// Mitsubishi GX Works2 project: SAPIR_SHELLY_FINAL   PLC: FX3G

// global labels: Global1
VAR_GLOBAL
  Start_Day_Light AT Y007 : BOOL;
  Input1 AT D1110 : REAL;
  Input2 AT D1120 : REAL;
  Input3 AT D1130 : REAL;
  Input4 AT D1140 : REAL;
  Raspberry AT D1115 : REAL;
  Lemon AT D1125 : REAL;
  Stability AT D1135 : REAL;
  Bears AT D1145 : REAL;
  Fin_inp AT M23 : BOOL;
  Startday AT X007 : BOOL;
  Stopday AT M27 : BOOL;
  AnalogOutput AT D8282 : INT;
  Package_Num AT D2000 : REAL;
  Emergency AT X005 : BOOL;
  Prepare_Flav AT X001 : BOOL;
  AnalogInput1 AT D8280 : INT;
END_VAR
VAR_GLOBAL CONSTANT
  Divide : REAL := 400.0;
END_VAR
VAR_GLOBAL
  DivOutput AT D1310 : REAL;
END_VAR
VAR_GLOBAL CONSTANT
  Regular_ice : REAL := 5.0;
END_VAR
VAR_GLOBAL
  Flav_Succeed AT M28 : BOOL;
  Regular_Chosen AT M30 : BOOL;
END_VAR
VAR_GLOBAL CONSTANT
  Needed1R : REAL := 280.0;
END_VAR
VAR_GLOBAL
  EnoughRas_R AT M29 : BOOL;
END_VAR
VAR_GLOBAL CONSTANT
  Needed2R : REAL := 455.0;
END_VAR
VAR_GLOBAL
  EnoughLem_R AT M40 : BOOL;
END_VAR
VAR_GLOBAL CONSTANT
  Needed3R : REAL := 105.0;
END_VAR
VAR_GLOBAL
  EnoughStab_R AT M41 : BOOL;
END_VAR
VAR_GLOBAL CONSTANT
  Needed4R : REAL := 28.0;
END_VAR
VAR_GLOBAL
  EnoughBear_R AT M42 : BOOL;
END_VAR
VAR_GLOBAL CONSTANT
  Needed1P : REAL := 385.0;
END_VAR
VAR_GLOBAL
  EnoughRas_P AT M45 : BOOL;
END_VAR
VAR_GLOBAL CONSTANT
  Needed2P : REAL := 665.0;
END_VAR
VAR_GLOBAL
  EnoughLem_P AT M48 : BOOL;
END_VAR
VAR_GLOBAL CONSTANT
  Needed3P : REAL := 210.0;
END_VAR
VAR_GLOBAL
  EnoughStab_P AT M50 : BOOL;
END_VAR
VAR_GLOBAL CONSTANT
  Needed4P : REAL := 70.0;
END_VAR
VAR_GLOBAL
  EnoughBear_P AT M52 : BOOL;
  Fin_Making_Light AT Y000 : BOOL;
  Timer_Making AT TS1 : BOOL;
  Making_Light AT Y000 : BOOL;
  Count_Yo AT TC1 : BOOL;
END_VAR
VAR_GLOBAL CONSTANT
  Fifty : INT := 50;
END_VAR
VAR_GLOBAL
  Next_Stage_Cool AT M60 : BOOL;
  Move_to_fridge AT X002 : BOOL;
  Fridge_Light AT Y002 : BOOL;
  Time_Of_Cool AT TS2 : BOOL;
  Sensor_Temp AT X003 : BOOL;
  Next_Stage_Mix AT M70 : BOOL;
  Flash_Y6 AT TS6 : BOOL;
  Flash_Y5 AT TS5 : BOOL;
  FlashLight_5 AT Y005 : BOOL;
  FlashLight_6 AT Y006 : BOOL;
  MixDone_R AT TS3 : BOOL;
  MixDone_P AT TS4 : BOOL;
  Pack_Done AT M90 : BOOL;
  Analogtemp AT D2020 : REAL;
  OutOfStock AT M20 : BOOL;
END_VAR
VAR_GLOBAL CONSTANT
  const_280 : REAL := 280.0;
END_VAR
VAR_GLOBAL
  Count_Y2 AT TC2 : BOOL;
END_VAR
VAR_GLOBAL CONSTANT
  Eighty : INT := 80;
END_VAR
VAR_GLOBAL
  Mixtime_R AT TC3 : BOOL;
END_VAR
VAR_GLOBAL CONSTANT
  Thirty : INT := 30;
END_VAR
VAR_GLOBAL
  Mixtime_P AT TC4 : BOOL;
  Hivhuv1 AT TC5 : BOOL;
END_VAR
VAR_GLOBAL CONSTANT
  Five : INT := 5;
END_VAR
VAR_GLOBAL
  Hivhuv2 AT TC6 : BOOL;
END_VAR
VAR_GLOBAL CONSTANT
  PlusOne : REAL := 1.0;
  fourty : REAL := 40.0;
END_VAR
VAR_GLOBAL
  TimeOfCooling AT TS2 : BOOL;
  Start_Y0 AT M62 : BOOL;
END_VAR
VAR_GLOBAL CONSTANT
  threehun5 : REAL := 350.0;
END_VAR
VAR_GLOBAL
  Making_Ras AT D1200 : REAL;
END_VAR
VAR_GLOBAL CONSTANT
  fortyhun9 : REAL := 490.0;
END_VAR
VAR_GLOBAL
  Making_Lem AT D1210 : REAL;
END_VAR
VAR_GLOBAL CONSTANT
  fifthhun6 : REAL := 560.0;
  sevenhun : REAL := 700.0;
END_VAR
VAR_GLOBAL
  Cooling_Ras AT D1220 : REAL;
  Cooling_Lem AT D1230 : REAL;
END_VAR
VAR_GLOBAL CONSTANT
  zero : REAL;
  zero2 : REAL;
  Eightsixeight : REAL := 868.0;
END_VAR
VAR_GLOBAL
  Mixing_All AT D1240 : REAL;
END_VAR
VAR_GLOBAL CONSTANT
  elefshlosmeot30 : REAL := 1330.0;
  elefshloshmeot30 : REAL := 1330.0;
END_VAR

// task Task_01 (event TRUE, interval 0, priority 31): POU_01

PROGRAM POU_01
(* structured ladder/FBD written out as ST: instructions are called as NAME(EN, inputs, outputs); _pN, _eN, _tN stand for wires *)
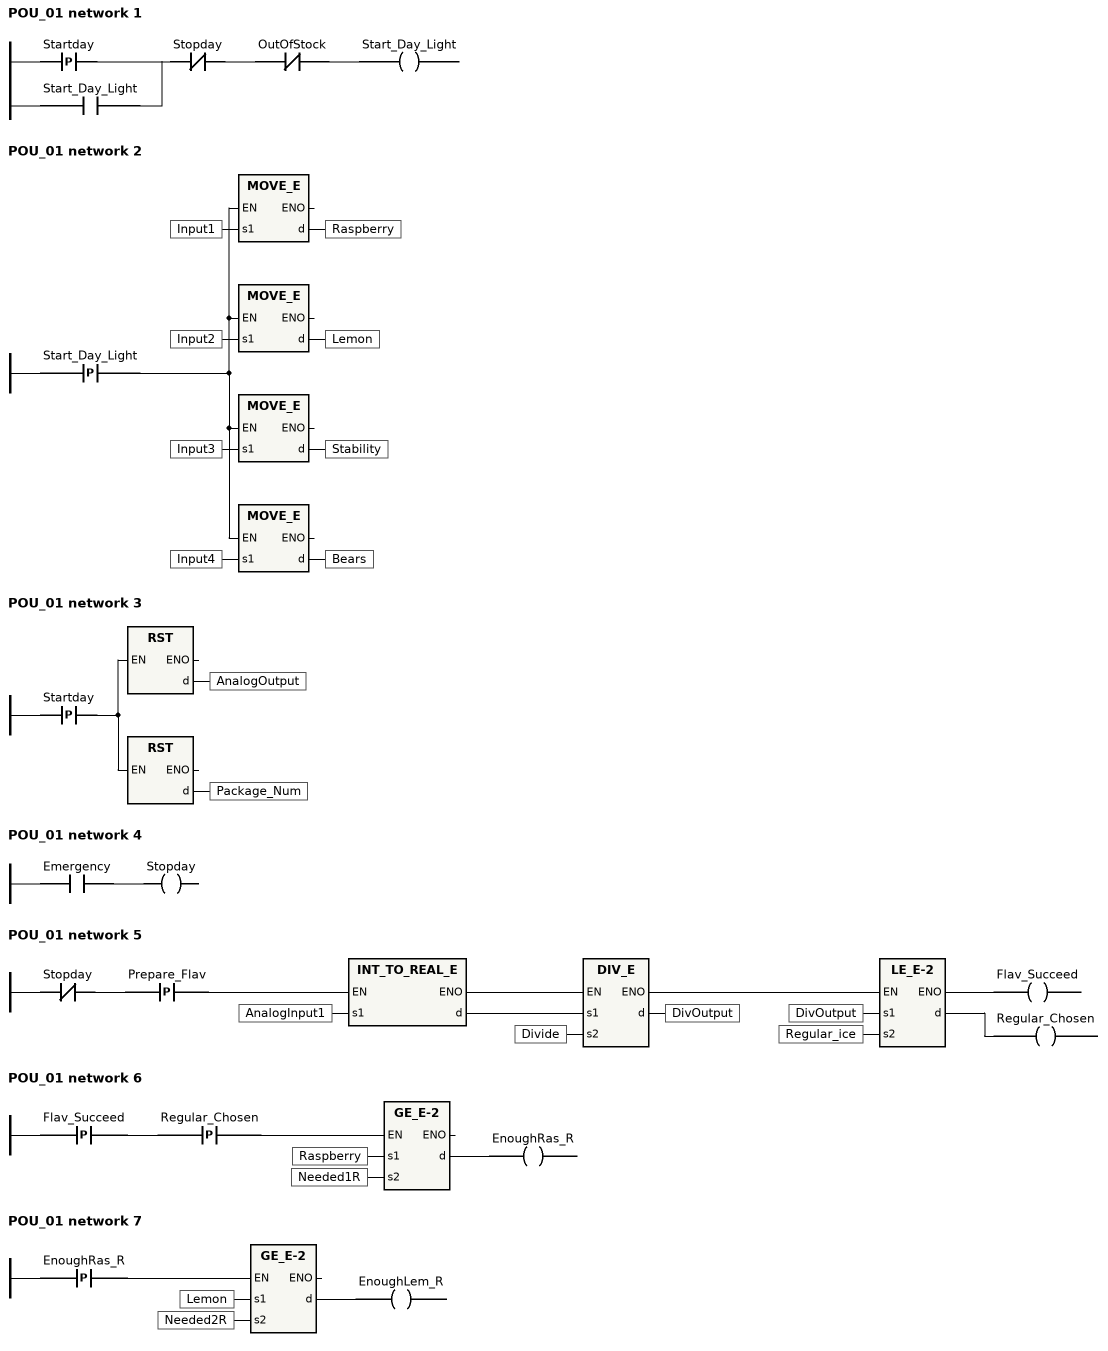
(* network 1 *)
Start_Day_Light := ((LDP(TRUE, Startday) OR Start_Day_Light) AND NOT Stopday) AND NOT OutOfStock;
(* network 2 *)
_p1 := LDP(TRUE, Start_Day_Light);
MOVE_E(_p1, Input1, Raspberry);
MOVE_E(_p1, Input2, Lemon);
MOVE_E(_p1, Input3, Stability);
MOVE_E(_p1, Input4, Bears);
(* network 3 *)
_p1 := LDP(TRUE, Startday);
RST(_p1, AnalogOutput);
RST(_p1, Package_Num);
(* network 4 *)
Stopday := Emergency;
(* network 5 *)
_e2 := INT_TO_REAL_E(NOT Stopday AND LDP(TRUE, Prepare_Flav), AnalogInput1, _t1);
_e3 := DIV_E(_e2, _t1, Divide, DivOutput);
_e5 := LE_E(_e3, DivOutput, Regular_ice, _t4);
Flav_Succeed := _e5;
Regular_Chosen := _t4;
(* network 6 *)
GE_E(LDP(TRUE, Flav_Succeed) AND LDP(TRUE, Regular_Chosen), Raspberry, Needed1R, _t1);
EnoughRas_R := _t1;
(* network 7 *)
GE_E(LDP(TRUE, EnoughRas_R), Lemon, Needed2R, _t1);
EnoughLem_R := _t1;
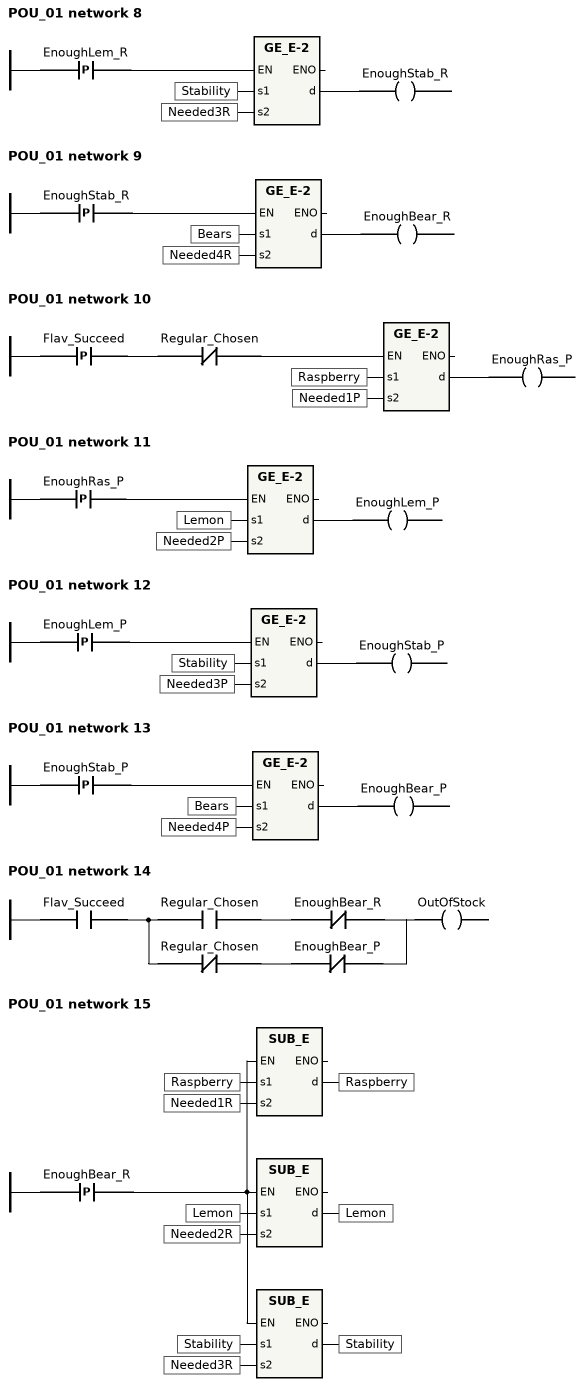
(* network 8 *)
GE_E(LDP(TRUE, EnoughLem_R), Stability, Needed3R, _t1);
EnoughStab_R := _t1;
(* network 9 *)
GE_E(LDP(TRUE, EnoughStab_R), Bears, Needed4R, _t1);
EnoughBear_R := _t1;
(* network 10 *)
GE_E(LDP(TRUE, Flav_Succeed) AND NOT Regular_Chosen, Raspberry, Needed1P, _t1);
EnoughRas_P := _t1;
(* network 11 *)
GE_E(LDP(TRUE, EnoughRas_P), Lemon, Needed2P, _t1);
EnoughLem_P := _t1;
(* network 12 *)
GE_E(LDP(TRUE, EnoughLem_P), Stability, Needed3P, _t1);
EnoughStab_P := _t1;
(* network 13 *)
GE_E(LDP(TRUE, EnoughStab_P), Bears, Needed4P, _t1);
EnoughBear_P := _t1;
(* network 14 *)
OutOfStock := (Flav_Succeed AND Regular_Chosen AND NOT EnoughBear_R) OR (Flav_Succeed AND NOT Regular_Chosen AND NOT EnoughBear_P);
(* network 15 *)
_p1 := LDP(TRUE, EnoughBear_R);
SUB_E(_p1, Raspberry, Needed1R, Raspberry);
SUB_E(_p1, Lemon, Needed2R, Lemon);
SUB_E(_p1, Stability, Needed3R, Stability);
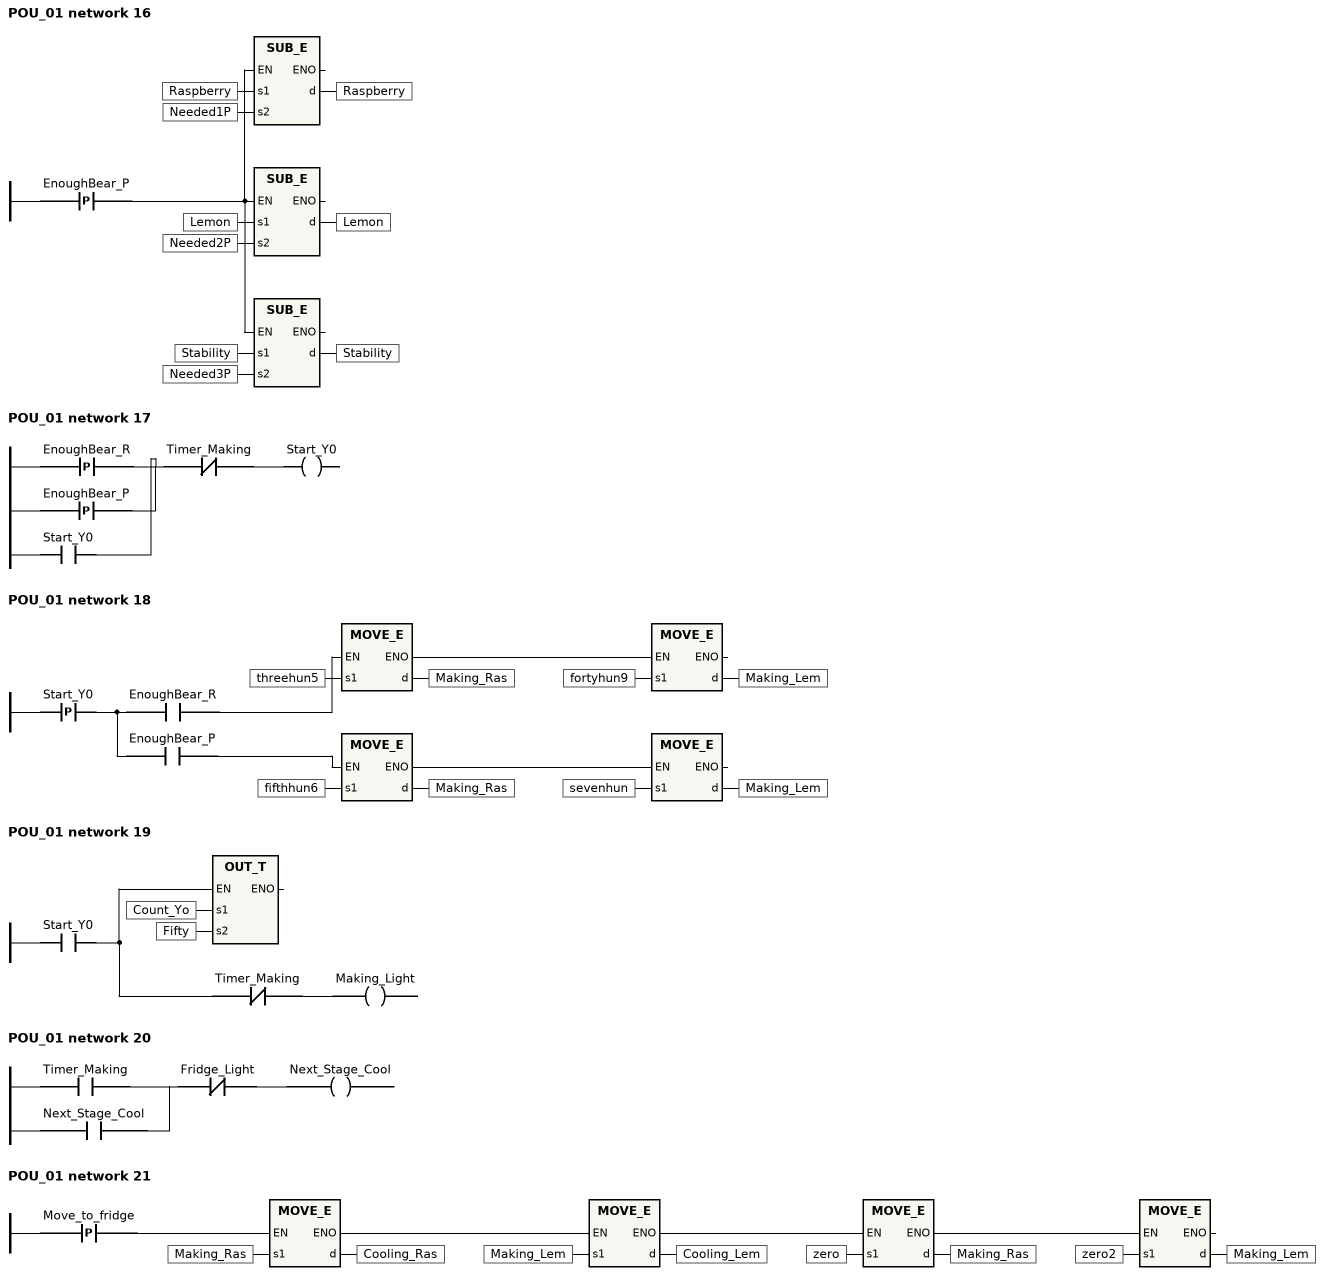
(* network 16 *)
_p1 := LDP(TRUE, EnoughBear_P);
SUB_E(_p1, Raspberry, Needed1P, Raspberry);
SUB_E(_p1, Lemon, Needed2P, Lemon);
SUB_E(_p1, Stability, Needed3P, Stability);
(* network 17 *)
Start_Y0 := (LDP(TRUE, EnoughBear_R) OR LDP(TRUE, EnoughBear_P) OR Start_Y0) AND NOT Timer_Making;
(* network 18 *)
_p1 := LDP(TRUE, Start_Y0);
_e2 := MOVE_E(_p1 AND EnoughBear_R, threehun5, Making_Ras);
MOVE_E(_e2, fortyhun9, Making_Lem);
_e3 := MOVE_E(_p1 AND EnoughBear_P, fifthhun6, Making_Ras);
MOVE_E(_e3, sevenhun, Making_Lem);
(* network 19 *)
OUT_T(Start_Y0, Count_Yo, Fifty);
Making_Light := Start_Y0 AND NOT Timer_Making;
(* network 20 *)
Next_Stage_Cool := (Timer_Making OR Next_Stage_Cool) AND NOT Fridge_Light;
(* network 21 *)
_e1 := MOVE_E(LDP(TRUE, Move_to_fridge), Making_Ras, Cooling_Ras);
_e2 := MOVE_E(_e1, Making_Lem, Cooling_Lem);
_e3 := MOVE_E(_e2, zero, Making_Ras);
MOVE_E(_e3, zero2, Making_Lem);
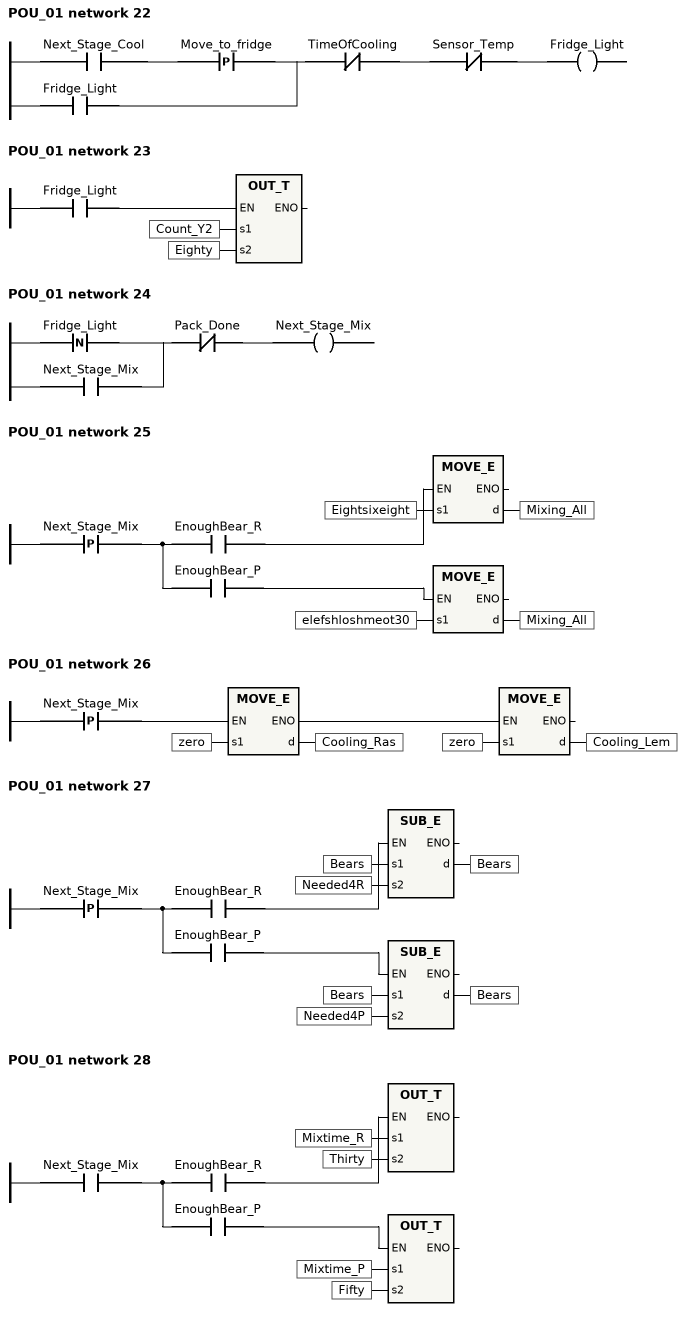
(* network 22 *)
Fridge_Light := (((Next_Stage_Cool AND LDP(TRUE, Move_to_fridge)) OR Fridge_Light) AND NOT TimeOfCooling) AND NOT Sensor_Temp;
(* network 23 *)
OUT_T(Fridge_Light, Count_Y2, Eighty);
(* network 24 *)
Next_Stage_Mix := (LDF(TRUE, Fridge_Light) OR Next_Stage_Mix) AND NOT Pack_Done;
(* network 25 *)
_p1 := LDP(TRUE, Next_Stage_Mix);
MOVE_E(_p1 AND EnoughBear_R, Eightsixeight, Mixing_All);
MOVE_E(_p1 AND EnoughBear_P, elefshloshmeot30, Mixing_All);
(* network 26 *)
_e1 := MOVE_E(LDP(TRUE, Next_Stage_Mix), zero, Cooling_Ras);
MOVE_E(_e1, zero, Cooling_Lem);
(* network 27 *)
_p1 := LDP(TRUE, Next_Stage_Mix);
SUB_E(_p1 AND EnoughBear_R, Bears, Needed4R, Bears);
SUB_E(_p1 AND EnoughBear_P, Bears, Needed4P, Bears);
(* network 28 *)
OUT_T(Next_Stage_Mix AND EnoughBear_R, Mixtime_R, Thirty);
OUT_T(Next_Stage_Mix AND EnoughBear_P, Mixtime_P, Fifty);
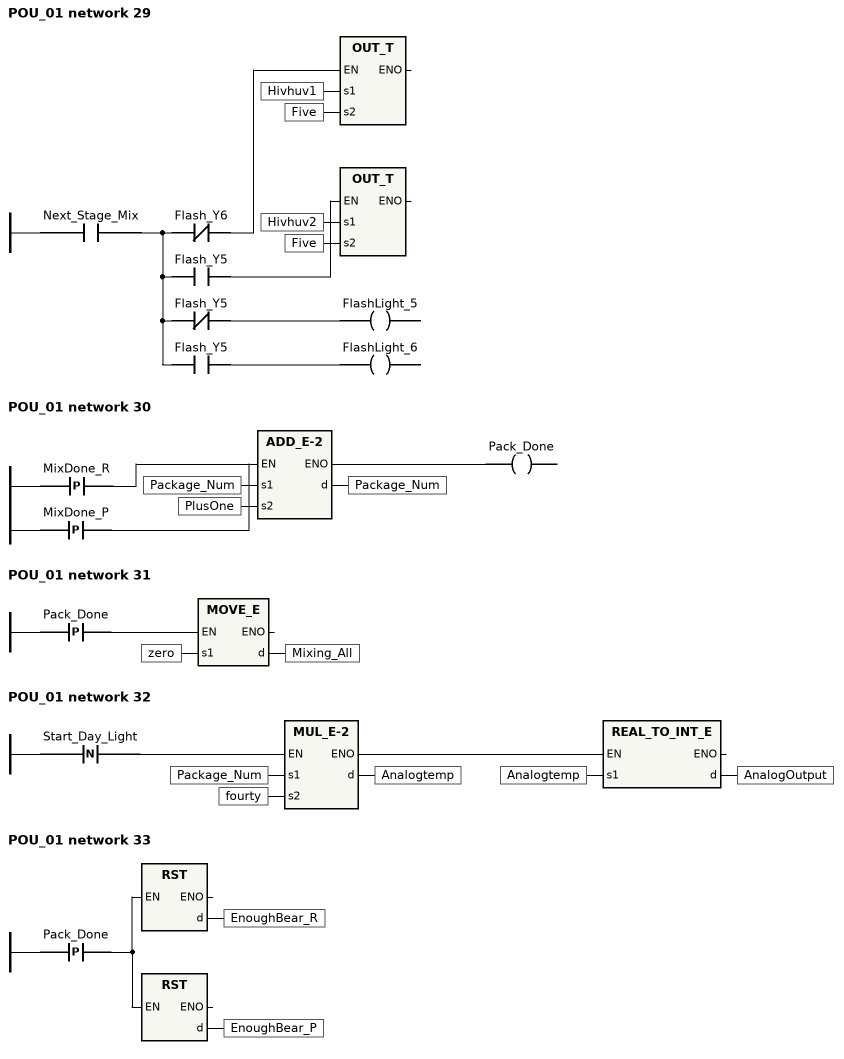
(* network 29 *)
OUT_T(Next_Stage_Mix AND NOT Flash_Y6, Hivhuv1, Five);
OUT_T(Next_Stage_Mix AND Flash_Y5, Hivhuv2, Five);
FlashLight_5 := Next_Stage_Mix AND NOT Flash_Y5;
FlashLight_6 := Next_Stage_Mix AND Flash_Y5;
(* network 30 *)
_e1 := ADD_E(LDP(TRUE, MixDone_R) OR LDP(TRUE, MixDone_P), Package_Num, PlusOne, Package_Num);
Pack_Done := _e1;
(* network 31 *)
MOVE_E(LDP(TRUE, Pack_Done), zero, Mixing_All);
(* network 32 *)
_e1 := MUL_E(LDF(TRUE, Start_Day_Light), Package_Num, fourty, Analogtemp);
REAL_TO_INT_E(_e1, Analogtemp, AnalogOutput);
(* network 33 *)
_p1 := LDP(TRUE, Pack_Done);
RST(_p1, EnoughBear_R);
RST(_p1, EnoughBear_P);
END_PROGRAM
